// TwinCAT 3 PLC project LogToFile
// Title: Logger
// Company: FCSL
// Author: FCSL
// ProjectVersion: 0.1.0.0
// Description: Logs and tracing
// ProgramVersion: 3.1.4026.13
// libraries:
//   SPT Base Types, * (Beckhoff Automation LLC)
//   SPT Components, * (Beckhoff Automation LLC)
//   Tc2_EtherCAT, * (Beckhoff Automation GmbH)
//   Tc2_Standard, * (Beckhoff Automation GmbH)
//   Tc2_System, * (Beckhoff Automation GmbH)
//   Tc2_Utilities, * (Beckhoff Automation GmbH)
//   Tc3_BA_Common, * (Beckhoff Automation GmbH)
//   Tc3_EventLogger, * (Beckhoff Automation GmbH)
//   Tc3_JsonXml, * (Beckhoff Automation GmbH)
//   TcUnit, * (www.tcunit.org)
//   VisuSymbols,3.5.10.0,System
// project tree:
//   DUTs/ E_Result.TcDUT
//   / GlobalTextList.TcGTLO, Logger.TcTTO, PlcTask.TcTTO, Visualization Manager.TcVMO (not stored)
//   Library/Emitter/KeyValueLog/AlarmLog/ FB_AlarmLog.TcPOU
//   Library/Emitter/KeyValueLog/AuditLog/ FB_AuditLog.TcPOU (not stored)
//   Library/Emitter/KeyValueLog/ FB_FCSLBaseKeyValueLog.TcPOU (not stored)
//   Library/Listener/KeyValueLog/AlarmLog/ FB_AlarmLogListener.TcPOU
//   Library/Listener/KeyValueLog/AuditLog/ FB_AuditLogListener.TcPOU
//   Library/Listener/KeyValueLog/ FB_FCSLBaseKeyValueLogListener.TcPOU, I_KeyValueLogListener.TcIO, ST_KeyValueLogMessage.TcDUT
//   Library/Listener/ PRG_Log_Main.TcPOU
//   Library/Listener/SysLog/ FB_SysLogListener.TcPOU, I_SysLogListener.TcIO, ST_SysLogMessages.TcDUT
//   Library/Emitter/ GVL_FCSLTracing.TcGVL
//   Library/Emitter/SysLog/ E_SysLogLevel.TcDUT, FB_SysLog.TcPOU
//   LogToFile/ E_LogToFile_State.TcDUT, FB_LogToFile.TcPOU, E_LogTransmittal.TcDUT, I_Logger.TcIO (not stored), ST_LoggerSettings.TcDUT
//   TestComponents/ FB_FCSLComponentBase.TcPOU
//   TestComponents/Test Components/ FB_Test_Component.TcPOU, I_TestComponent.TcIO, PRG_TestComponents.TcPOU
//   POUs/ FB_AppendToFileDaily.TcPOU, PRG_Main.TcPOU
//   Version/ Global_Version.TcGVL
// real-time tasks:
//   TASK PlcTask: cycle T#50000us, priority 8, ADS port 350
//   TASK Logger: cycle T#10ms, priority 6, ADS port 351

CONFIGURATION LogToFile
    RESOURCE PLC ON TwinCAT3
        TASK Logger(INTERVAL := T#10ms, PRIORITY := 6);
        TASK PlcTask(INTERVAL := T#50000us, PRIORITY := 8);
        PROGRAM PRG_Log_Main WITH Logger : PRG_Log_Main;
        PROGRAM PRG_TestComponents WITH PlcTask : PRG_TestComponents;
    END_RESOURCE
END_CONFIGURATION

// ---- DUTs/E_Result.TcDUT
{attribute 'qualified_only'}
{attribute 'strict'}
{attribute 'to_string'}
TYPE E_Result :
(
	invalid := 0,
	inProgress,
	done,
	aborted
);
END_TYPE

// ---- Library/Listener/KeyValueLog/ST_KeyValueLogMessage.TcDUT
TYPE ST_KeyValueLogMessage :
    STRUCT
        timestamp 	: T_MaxString;
        k   		: T_MaxString;
        v   		: T_MaxString;	
    END_STRUCT
END_TYPE

// ---- Library/Listener/SysLog/ST_SysLogMessages.TcDUT
TYPE ST_SysLogMessages :
    STRUCT
        Timestamp : T_MaxString;
        Message   : T_MaxString;
	    LogLevel  : E_SysLogLevel;
		Source    : T_MaxString;
        Context   : T_MaxString;
        ScanCount : UDINT;
        Flags     : UDINT;
		Json   : T_MaxString;
    END_STRUCT
END_TYPE

// ---- Library/Emitter/SysLog/E_SysLogLevel.TcDUT
{attribute 'qualified_only'}
{attribute 'to_string'}
TYPE E_SysLogLevel :
(
	invalid := 0,
	testing,
	commissioning,
	production
) UDINT;
END_TYPE

// ---- LogToFile/E_LogToFile_State.TcDUT
{attribute 'qualified_only'}
{attribute 'strict'}
TYPE E_LogToFile_State :
(
	IDLE, 
	PREPARE_DATA, 
	OPEN_FILE, 
	WRITE_TO_FILE, 
	CLOSE_FILE, 
	RESET
);
END_TYPE

// ---- LogToFile/E_LogTransmittal.TcDUT
{attribute 'qualified_only'}
{attribute 'strict'}
{attribute 'to_string'}
TYPE E_LogTransmittal :
(
	invalid := 0,
	toFile,
	viaMQTT,
	viaHTTP,
	viaWS
);
END_TYPE

// ---- LogToFile/ST_LoggerSettings.TcDUT
TYPE ST_LoggerSettings :
STRUCT
	netID : STRING(20);
	filePath : T_MaxString;
	filePrefix : STRING(10);
	FileType : STRING(10);
END_STRUCT
END_TYPE

// ---- Library/Emitter/GVL_FCSLTracing.TcGVL
{attribute 'qualified_only'}
VAR_GLOBAL
	// System Log [Saved to Disk]
	sysLogLevel 		: E_SysLogLevel := E_SysLogLevel.testing;  // Current level to log to file	
	sysLog 				: FB_SysLog;
	
	// Audit Log
	auditLog 			: FB_AuditLog;
	
	//Alarm Log
	alarmLog			: FB_AlarmLog;
END_VAR

// ---- Version/Global_Version.TcGVL
{attribute 'TcGenerated'}
{attribute 'no-analysis'}
{attribute 'linkalways'}
// This function has been automatically generated from the project information.
VAR_GLOBAL CONSTANT
	{attribute 'const_non_replaced'}
	stLibVersion_Logger : ST_LibVersion := (iMajor := 0, iMinor := 1, iBuild := 0, iRevision := 0, nFlags := 0, sVersion := '0.1.0.0');
END_VAR

// ---- Library/Listener/KeyValueLog/I_KeyValueLogListener.TcIO
INTERFACE I_KeyValueLogListener

METHOD OnTraceReceived
VAR_INPUT
    message : ST_KeyValueLogMessage;
END_VAR
END_METHOD

END_INTERFACE

// ---- Library/Listener/SysLog/I_SysLogListener.TcIO
INTERFACE I_SysLogListener

METHOD OnTraceReceived
VAR_INPUT
    message : ST_SysLogMessages;
END_VAR
END_METHOD

END_INTERFACE

// ---- TestComponents/Test Components/I_TestComponent.TcIO
INTERFACE I_TestComponent EXTENDS I_BaseFB

END_INTERFACE

// ---- Library/Listener/PRG_Log_Main.TcPOU
PROGRAM PRG_Log_Main

VAR
	sysLogger 		: FB_SysLogListener;
	auditLogger		: FB_AuditLogListener;
	alarmLogger		: FB_AlarmLogListener;
END_VAR

sysLogger.CyclicLogic();
auditLogger.CyclicLogic();
alarmLogger.CyclicLogic();

END_PROGRAM

// ---- Library/Listener/SysLog/FB_SysLogListener.TcPOU
FUNCTION_BLOCK FB_SysLogListener EXTENDS FB_ListenerBase2 IMPLEMENTS I_SysLogListener
VAR
    json          			: FB_JsonDomParser; 		//Parse JSON attribute of messages
    jsonAttribute 			: STRING(10000);    		//Holds JSON attribute
    hr           			: HRESULT;         		//Signals JSON attribute was successfully read
    ipListener    			: I_SysLogListener; 	//Receives callback once message is processed
	
	fbRequestEventText 		: FB_RequestEventText;
	{attribute 'TcEncoding':='UTF-8'}
	sLastMessageText 		: STRING;
	
	
	_InitComplete			: BOOL;
	
	logger 					: FB_LogToFile;
END_VAR

METHOD CyclicLogic
IF ( NOT _initComplete ) THEN
    _initComplete := Initialize();
    RETURN;
END_IF

Execute();

logger.CyclicLogic();
END_METHOD

METHOD Initialize : BOOL
VAR
    listenerFilter 		: FB_TcEventFilter;
    hr             		: HRESULT;
END_VAR
Listener := THIS^;                                   //For callbacks on message received
ListenerFilter.Clear().EventClass.EqualTo(TC_EVENT_CLASSES.SysLog); //Filter events by tracing class
hr := Subscribe2(ListenerFilter);                    //Subscribe to retrieve defined events
IF ( SUCCEEDED(hr) ) THEN
    Initialize := TRUE;
END_IF
END_METHOD

PROPERTY Listener : I_SysLogListener
SET
ipListener := Listener;
END_SET
END_PROPERTY

METHOD OnMessageSent : Tc3_EventLogger.HRESULT
VAR_INPUT
    fbEvent 			: REFERENCE TO FB_TcEvent;
END_VAR

VAR
    message      		: ST_SysLogMessages;
    jsonDocument 		: SJsonValue;
    jsonProperty 		: SJsonValue;
	
	hasMember 			: BOOL;
END_VAR
hr := fbEvent.GetJsonAttribute(JsonAttribute, SIZEOF(JsonAttribute));

IF ( SUCCEEDED(hr) ) THEN
    jsonDocument := json.ParseDocument(JsonAttribute);

    IF ( json.HasMember(jsonDocument, 'Timestamp') ) THEN
        jsonProperty      := json.FindMember(JsonDocument, 'Timestamp');
        message.timestamp := json.GetString(JsonProperty);
    END_IF

    IF ( json.HasMember(jsonDocument, 'Message') ) THEN
        jsonProperty    := json.FindMember(jsonDocument, 'Message');
        message.message := json.GetString(jsonProperty);
    END_IF
	
	IF ( json.HasMember(jsonDocument, 'LogLevel') ) THEN
        jsonProperty      := json.FindMember(jsonDocument, 'LogLevel');
        message.logLevel := json.GetUint(jsonProperty);
    END_IF
	
    IF ( json.HasMember(jsonDocument, 'Source') ) THEN
        jsonProperty   := json.FindMember(jsonDocument, 'Source');
        message.Source := json.GetString(jsonProperty);
    END_IF

    IF ( json.HasMember(jsonDocument, 'Context') ) THEN
        jsonProperty    := json.FindMember(jsonDocument, 'Context');
        message.Context := json.GetString(jsonProperty);
    END_IF

    IF ( json.HasMember(jsonDocument, 'ScanCount') ) THEN
        jsonProperty      := json.FindMember(jsonDocument, 'ScanCount');
        message.ScanCount := json.GetUint(jsonProperty);
    END_IF

    IF ( json.HasMember(jsonDocument, 'Flags') ) THEN
        jsonProperty  := json.FindMember(jsonDocument, 'Flags');
        message.Flags := json.GetUint(jsonProperty);
    END_IF
	
    IF ( json.HasMember(jsonDocument, 'ExtendedInfo') ) THEN
        jsonProperty := json.FindMember(jsonDocument, 'ExtendedInfo');
        message.Json := json.GetString(jsonProperty);
    END_IF


    IF ( ipListener <> 0 ) THEN
        //Notify listener of message data
        ipListener.OnTraceReceived(Message);
    END_IF
END_IF

OnMessageSent := S_OK; // in order to receive more callbacks (Set <> S_OK in order to cancel the callbacks for this program cycle.)]]>
END_METHOD

METHOD OnTraceReceived
VAR_INPUT
    message 			: ST_SysLogMessages;
END_VAR

VAR
	timestamp 			: T_MaxString;
	msg   				: T_MaxString;
	logLevel  			: E_SysLogLevel;
	source    			: T_MaxString;
	context   			: T_MaxString;
	scanCount 			: UDINT;
	flags     			: UDINT;
END_VAR
// Extract relevant fields
timestamp := message.Timestamp;
msg   	  := message.Message;
logLevel  := message.LogLevel;
source    := message.Source;
context   := message.Context;
scanCount := message.ScanCount;
flags     := message.Flags;


logger.M_AddSysLog(1,msg);
END_METHOD

END_FUNCTION_BLOCK

// ---- LogToFile/FB_LogToFile.TcPOU
FUNCTION_BLOCK FB_LogToFile EXTENDS FB_CyclicFB

VAR CONSTANT
	LOG_SETTINGS 				: ST_LoggerSettings := (netID := '', filePath := 'C:\Logs\', filePrefix := 'SystemApp_', FileType := '.txt');	
	LOG_TIMEOUT 				: TIME := T#5S;
	EXPORT_INTERVAL				: TIME := T#10S;
	NEW_LINE 					: STRING(2) := '$r$n'; // Newline character
END_VAR

VAR
    ringBuffer 					: FB_StringRingBuffer;
    bufferMemory 				: ARRAY[0..5000] OF BYTE; // Adjust size as needed
	
	firstCycle 					: BOOL := TRUE;
	exportTimer					: TON;
	
	// From FB_init
    _netId 	 					: T_AmsNetId;     // Net ID for file operations
    _dirPath 					: T_MaxString;    // Directory path for the log file
	_logPrefix  				: STRING(10);     // Prefix for log file
	_fileExtension 				: STRING(10);  // File extension i.e. '.txt'
	_timeOut 					: TIME := DEFAULT_ADS_TIMEOUT;

// Params
	_execute 					: BOOL := FALSE; // Trigger for the log operation
    _data 	 					: T_MaxString; // Log entry to write

// Internal
	state 						: E_LogToFile_State;

    fileOpen  					: FB_FileOpen;
    fileClose 					: FB_FileClose;
    fileWrite 					: FB_FileWrite;

	fileRef 					: UINT := 0;       	// File handle
    risingEdge 					: R_TRIG;     // Rising edge detector for execute signal
END_VAR

VAR_OUTPUT
	smDone, smBusy, smError : BOOL;
    errId : UDINT;	 // Error ID in case of failure
END_VAR

METHOD CyclicLogic
VAR
	bufferFillPercentage: UDINT;
END_VAR
IF ( firstCycle ) THEN
	ringBuffer( pBuffer := ADR(bufferMemory), cbBuffer := SIZEOF(bufferMemory), bOverwrite := TRUE );
	firstCycle := FALSE;
	state := E_LogToFile_State.IDLE;
	RETURN;
END_IF

ringBuffer();

exportTimer(IN := TRUE, PT := EXPORT_INTERVAL);
bufferFillPercentage := (ringBuffer.cbSize * 100) / SIZEOF(bufferMemory);

IF ( ( exportTimer.Q  ) AND ( ringBuffer.nCount > 0 ) ) OR (bufferFillPercentage > 50) THEN
	//M_WriteToFile(); // Export logs when conditions are met
	_execute := TRUE;
	exportTimer(IN := FALSE); // Reset timer
ELSE
	_execute := FALSE;
END_IF;

M_StateMachine();
END_METHOD

//FB_Init is always available implicitly and it is used primarily for initialization.
//The return value is not evaluated. For a specific influence, you can also declare the
//methods explicitly and provide additional code there with the standard initialization
//code. You can evaluate the return value.
METHOD FB_Init: BOOL
VAR_INPUT
    bInitRetains: BOOL; // TRUE: the retain variables are initialized (reset warm / reset cold)
    bInCopyCode: BOOL;  // TRUE: the instance will be copied to the copy code afterward (online change)
END_VAR
_netID := LOG_SETTINGS.netID;
_dirPath := LOG_SETTINGS.filePath;
_logPrefix := LOG_SETTINGS.filePrefix;
_fileExtension := LOG_SETTINGS.FileType;
_timeOut := LOG_TIMEOUT;
END_METHOD

METHOD M_AddKeyValueLog : BOOL

VAR_INPUT
    message : ST_KeyValueLogMessage;
END_VAR

VAR
    logEntry : STRING;
END_VAR
// Concatenate severity and message
logEntry := CONCAT(message.k, ' - ');
logEntry := CONCAT(logEntry, message.v);
logEntry := CONCAT(logEntry, ' at ');
logEntry := CONCAT(logEntry, message.timestamp);

// Add log entry to ring buffer
ringBuffer.A_AddTail(putValue := logEntry);
IF ( NOT ringbuffer.bOk ) THEN
	// Handle write error (optional)END_IF;
END_IF
END_METHOD

METHOD PUBLIC M_AddSysLog : BOOL

VAR_INPUT
    severity : INT;
    message : STRING;
END_VAR

VAR
    logEntry : STRING;
END_VAR
// Concatenate severity and message
logEntry := CONCAT('Severity ', INT_TO_STRING(severity));
logEntry := CONCAT(logEntry, ': ');
logEntry := CONCAT(logEntry, message);

// Add log entry to ring buffer
ringBuffer.A_AddTail(putValue := logEntry);
IF ( NOT ringbuffer.bOk ) THEN
	// Handle write error (optional)END_IF;
END_IF
END_METHOD

METHOD PRIVATE M_CloseFile : BOOL

VAR_INPUT
	execute : BOOL;	
END_VAR
IF ( NOT execute ) THEN
	fileOpen(bExecute := FALSE);
	M_CloseFile := FALSE;
	RETURN;
END_IF

IF ( NOT fileOpen.bBusy ) THEN     
	fileClose(sNetId := _netId, hFile := fileRef, tTimeout := _timeOut);
END_IF

// Attempt to close the file
fileClose(bExecute := TRUE);

IF ( NOT M_HandleError(fileClose.bError , fileClose.nErrId) ) THEN
	fileRef := 0; // File handle
END_IF

M_CloseFile := fileClose.bBusy;
END_METHOD

METHOD PRIVATE M_HandleError : BOOL
VAR_INPUT
	check 					: BOOL;
	errorID 				: UDINT;
END_VAR
check := error;

IF check THEN
	errId := errorID;
END_IF

M_HandleError := check;
END_METHOD

METHOD PRIVATE M_OpenFile : BOOL

VAR_INPUT
	execute 				: BOOL;	
END_VAR

VAR
	getSystemTime 			: GETSYSTEMTIME; // System time function block
	fileTime 				: T_FILETIME;     // File time
	dateString 				: STRING;		// Date string for filename
	filePath 				: STRING; 	// Full log file path
END_VAR
IF ( NOT execute ) THEN
	fileOpen(bExecute := FALSE);
	M_OpenFile := FALSE;
	RETURN;
END_IF

IF ( _dirPath = '' ) THEN
   	M_HandleError(TRUE , 99);
	M_OpenFile := FALSE;
    RETURN;
END_IF

IF ( NOT fileOpen.bBusy ) THEN
	// Generate log file path with current date
	getSystemTime(timeLoDW => fileTime.dwLowDateTime, timeHiDW => fileTime.dwHighDateTime );
	dateString := SYSTEMTIME_TO_STRING(FILETIME_TO_SYSTEMTIME(fileTime));
	filepath := CONCAT(_dirPath, _logPrefix); 			// Create file path
	filePath := CONCAT(filepath, LEFT(dateString, 10)); // Add date to file path
	filePath := CONCAT(filepath, _fileExtension); 		// Add file extension to file path.
     
	fileOpen(sNetId := '', sPathName := filePath, nMode := FOPEN_MODEAPPEND, ePath := PATH_GENERIC, tTimeout := _timeOut);
END_IF

// Attempt to open the file
fileOpen(bExecute := TRUE);

IF ( NOT M_HandleError(fileOpen.bError , fileOpen.nErrId) ) THEN
	fileRef := fileOpen.hFile; // No error case
END_IF

M_OpenFile := fileOpen.bBusy;
END_METHOD

METHOD M_StateMachine

VAR
	status			: BOOL;
END_VAR
RisingEdge(CLK := _execute);

CASE state OF
    E_LogToFile_State.IDLE: // Idle state
        IF ( RisingEdge.Q ) THEN
			smDone := FALSE;
           	smBusy := TRUE;
            smError := FALSE;
            errId := 0;
		
			fileOpen(bExecute := FALSE);
			fileWrite(bExecute := FALSE);
			fileClose(bExecute := FALSE);

            state := E_LogToFile_State.OPEN_FILE;
        END_IF

    E_LogToFile_State.OPEN_FILE: // Open the file
        status := M_OpenFile(TRUE);
		IF error THEN
			state := E_LogToFile_State.CLOSE_FILE;
        ELSIF ( fileRef <> 0 ) AND ( NOT status ) THEN
			M_OpenFile(FALSE);
			state := E_LogToFile_State.PREPARE_DATA;
        END_IF
		
	E_LogToFile_State.PREPARE_DATA:
		ringBuffer.A_RemoveHead();
		_data := ringBuffer.getValue;
		
		IF ( _data <> '' ) THEN
			M_WriteToFile(FALSE, '');
			state := E_LogToFile_State.WRITE_TO_FILE;
		ELSE
			IF ( NOT fileWrite.bBusy ) THEN
				state := E_LogToFile_State.CLOSE_FILE;
			END_IF
		END_IF
		
    E_LogToFile_State.WRITE_TO_FILE: // Write to the file
		status := M_WriteToFile(execute := TRUE, inputString := _data);
		
		IF ( NOT status ) THEN
			state := E_LogToFile_State.PREPARE_DATA;
		END_IF
	
    
    E_LogToFile_State.CLOSE_FILE: // Close the file
       IF ( fileREF <> 0 ) THEN
			status :=  M_CloseFile(TRUE);
			IF ( error OR ( NOT fileWrite.bBusy ) ) THEN
				M_CloseFile(FALSE);
				state := E_LogToFile_State.RESET;
        	END_IF
		ELSE
			M_CloseFile(FALSE);
			state := E_LogToFile_State.RESET;
	   END_IF

    E_LogToFile_State.RESET: // Cleanup and reset
		smDone := TRUE;
		smBusy := FALSE;
        fileRef := 0;;
        state := E_LogToFile_State.IDLE; // Return to idle state
END_CASE
END_METHOD

METHOD PRIVATE M_WriteToFile : BOOL

VAR_INPUT
	execute : BOOL;
	inputString : STRING; // Log entry to write
END_VAR

VAR
	msgString : STRING;
END_VAR
IF ( NOT execute ) THEN
	fileOpen(bExecute := FALSE);
	fileWrite(bExecute := FALSE);
	M_WriteToFile := FALSE;
	RETURN;
END_IF

IF ( NOT fileWrite.bBusy ) THEN
	
	IF ( LEN(inputString) > (UINT_TO_INT(SIZEOF(msgString)) - LEN(NEW_LINE))) THEN
		M_HandleError( TRUE, 98);
		M_WriteToFile := FALSE;
		RETURN;
	END_IF

	msgString := CONCAT( inputString, NEW_LINE );

	// Write the message to the file
	fileWrite(sNetId := _netId, hFile := fileRef, pWriteBuff := ADR(msgString), cbWriteLen := INT_TO_UDINT(LEN(msgString)), tTimeout := +_timeOut);
END_IF

// Attempt to write the file
fileWrite(bExecute := TRUE);

IF ( M_HandleError(fileWrite.bError , fileWrite.nErrId) ) THEN
	M_WriteToFile := FALSE; // File handle
	RETURN;
END_IF

M_WriteToFile := fileWrite.bBusy;
END_METHOD

END_FUNCTION_BLOCK

// ---- Library/Listener/KeyValueLog/AuditLog/FB_AuditLogListener.TcPOU
FUNCTION_BLOCK FB_AuditLogListener EXTENDS FB_FCSLBaseKeyValueLogListener

METHOD Initialize : BOOL
VAR
    ListenerFilter : FB_TcEventFilter;
    hr             : HRESULT;
END_VAR
Listener := THIS^;                                   //For callbacks on message received
ListenerFilter.Clear().EventClass.EqualTo(TC_EVENT_CLASSES.AuditLog); //Filter events by tracing class
hr := Subscribe2(ListenerFilter);                    //Subscribe to retrieve defined events
IF ( SUCCEEDED(hr) ) THEN
    Initialize := TRUE;
END_IF
END_METHOD

END_FUNCTION_BLOCK

// ---- Library/Listener/KeyValueLog/FB_FCSLBaseKeyValueLogListener.TcPOU
FUNCTION_BLOCK FB_FCSLBaseKeyValueLogListener EXTENDS FB_ListenerBase2 IMPLEMENTS I_KeyValueLogListener
VAR
    json          			: FB_JsonDomParser; 		//Parse JSON attribute of messages
    jsonAttribute 			: STRING(10000);    		//Holds JSON attribute
    hr           			: HRESULT;         		//Signals JSON attribute was successfully read
    ipListener    			: I_KeyValueLogListener; 	//Receives callback once message is processed
	
	fbRequestEventText 		: FB_RequestEventText;
	{attribute 'TcEncoding':='UTF-8'}
	sLastMessageText 		: STRING;
	
	
	_initComplete			: BOOL;
	
	logger 					: FB_LogToFile;
END_VAR

METHOD CyclicLogic
IF NOT _InitComplete THEN
    _InitComplete := Initialize();
    RETURN;
END_IF

Execute();

logger.CyclicLogic();
END_METHOD

METHOD Initialize : BOOL
END_METHOD

PROPERTY Listener : I_KeyValueLogListener
SET
ipListener := Listener;
END_SET
END_PROPERTY

METHOD OnMessageSent : Tc3_EventLogger.HRESULT
VAR_INPUT
    fbEvent 			: REFERENCE TO FB_TcEvent;
END_VAR

VAR
    message      		: ST_KeyValueLogMessage;
    jsonDocument 		: SJsonValue;
    jsonProperty 		: SJsonValue;
	jsonExtendedInfo	: SJsonValue;
	
	bHasMember 			: BOOL;
END_VAR
hr := fbEvent.GetJsonAttribute(JsonAttribute, SIZEOF(JsonAttribute));

IF ( SUCCEEDED(hr) ) THEN
    jsonDocument := json.ParseDocument(jsonAttribute);

    IF ( json.HasMember(jsonDocument, 'Timestamp') ) THEN
        jsonProperty      := json.FindMember(jsonDocument, 'Timestamp');
        message.Timestamp := json.GetString(jsonProperty);
    END_IF

    IF ( json.HasMember(jsonDocument, 'k') ) THEN
        jsonProperty    := json.FindMember(jsonDocument, 'k');
        message.k := json.GetString(jsonProperty);
    END_IF
	
    IF ( json.HasMember(jsonDocument, 'v') ) THEN
        jsonProperty    := json.FindMember(jsonDocument, 'v');
 		message.v := json.GetString(jsonProperty);
    END_IF

    IF ( ipListener <> 0 ) THEN
        //Notify listener of message data
        ipListener.OnTraceReceived(Message);
    END_IF
END_IF

OnMessageSent := S_OK; // in order to receive more callbacks (Set <> S_OK in order to cancel the callbacks for this program cycle.)
END_METHOD

METHOD OnTraceReceived
VAR_INPUT
    message : ST_KeyValueLogMessage;
END_VAR

VAR
	timestamp			: Tc2_System.T_MaxString;
	key					: Tc2_System.T_MaxString;
	value				: Tc2_System.T_MaxString;
END_VAR
// Extract relevant fields
timestamp   := message.Timestamp;
key   := message.k;
value   := message.v;

logger.M_AddKeyValueLog(message);
END_METHOD

END_FUNCTION_BLOCK

// ---- Library/Listener/KeyValueLog/AlarmLog/FB_AlarmLogListener.TcPOU
FUNCTION_BLOCK FB_AlarmLogListener EXTENDS FB_FCSLBaseKeyValueLogListener

METHOD Initialize : BOOL
VAR
    ListenerFilter : FB_TcEventFilter;
    hr             : HRESULT;
END_VAR
Listener := THIS^;                                   //For callbacks on message received
ListenerFilter.Clear().EventClass.EqualTo(TC_EVENT_CLASSES.AlarmLog); //Filter events by tracing class
hr := Subscribe2(ListenerFilter);                    //Subscribe to retrieve defined events
IF ( SUCCEEDED(hr) ) THEN
    Initialize := TRUE;
END_IF
END_METHOD

END_FUNCTION_BLOCK

// ---- TestComponents/Test Components/PRG_TestComponents.TcPOU
PROGRAM PRG_TestComponents
VAR
	// Interfaces
	iComponent1, iComponet2, iComponet3 : I_TestComponent;	

	// Componentes
	Component_1 : FB_Test_Component := (Name := 'TC-01');
	Component_2 : FB_Test_Component := (Name := 'TC-02');
	Component_3 : FB_Test_Component := (Name := 'TC-03');

	// Test Triggers
	Trig1a, Trig1b, Trig2a, Trig2b, Trig3a, Trig3b : BOOL;
END_VAR

M_Map();

METHOD M_Map : BOOL
VAR_INPUT
END_VAR
// Map Interface
iComponent1 := Component_1;
iComponet2 := Component_2;
iComponet3 := Component_3;

// Map Parameters
Component_1.pTrig := Trig1a;
Component_1.pTrig2 := Trig1b;
Component_2.pTrig := Trig2a;
Component_2.pTrig2 := Trig2b;
Component_3.pTrig := Trig3a;
Component_3.pTrig2 := Trig3b;

// Cylic Calls
Component_1.M_CyclicLogic();
Component_2.M_CyclicLogic();
Component_3.M_CyclicLogic();
END_METHOD

END_PROGRAM

// ---- TestComponents/Test Components/FB_Test_Component.TcPOU
FUNCTION_BLOCK FB_Test_Component EXTENDS FB_FCSLComponentBase IMPLEMENTS I_TestComponent

VAR
	_trig : BOOL;
	Trig : R_TRIG;
	_trig2 : BOOL;
	Trig2 : R_TRIG;
END_VAR

VAR
	// Inputs
	MyInput AT %I* : BOOL;

	// Outputs
	MyOutput AT %Q* : BOOL;

	// HMI
//	MyComponent_HMI			: ST_ComponentMyComponent_HMI;
//	HMICommandDescendant_RT : R_TRIG;

	// Alarms
//	MyComponentAlarms : ARRAY[1..MY_COMPONENT_ALARMS_COUNT] OF FB_TcAlarm;

	// Internal variables
//	_MyVarProperty1 : BOOL;
//	_MyVarProperty2 : BOOL;
//	MyVarInternal1	: BOOL;
//	MyVarInternal2	: BOOL;

	//MyCommandFb		: MyCommandFB;// Command FB to execute something e.g. MC_MoveAbsolute
END_VAR

VAR CONSTANT
//	MY_COMPONENT_ALARMS_COUNT : UDINT := 2;
END_VAR

// NO CODE HERE!!!

//! @summary Basic component initialization logic
METHOD PRIVATE CyclicLogic

//! @description This method is called by <c>CyclicLogic()</c> as required
//! @description This method should be called cyclically by descendant function blocks by invoking <c>SUPER^.CyclicLogic()</c>. 
// Alternatively, the contents of this method could be reimplemented entirely in which case a call to this method would not be necessary.

VAR
END_VAR
IF NOT _InitComplete THEN
	_InitComplete := Initialize();
	RETURN;
END_IF

//{error 'Programming instruction - Write your custom component cyclic cogic here'}

Trig(CLK := _trig);
Trig2(CLK := _trig2);

IF Trig.Q THEN
	M_SysLog(msg := CONCAT(Name, ' : Has being triggered 1'), debug := E_SysLogLevel.testing);
END_IF

IF Trig.Q THEN
	M_AlarmLog(k := 'Raised', v := 'PT-05 warning raised, value: 5555');
END_IF
IF Trig2.Q THEN
	M_AuditLog(k := 'Login', v := 'User 1234 has logged in');
END_IF

(*
	MyCommandFb();
	IF MyCommandFB.Error THEN
		_Error	 := TRUE;
		_ErrorID := MyCommandFb.ErrorId;
	END_IF
	
	MyCommandFB.Execute := FALSE;
*)

// Component Error
//{error 'Programming instruction - Create component has error'}
//_Error	 := TRUE;
//_ErrorID := 9999;

// Component Busy
//{error 'Programming instruction - Create component is busy'}
IF FALSE THEN
	_Busy := TRUE;
ELSE
	_Busy := FALSE;
END_IF

// Call Super
SUPER^.CyclicLogic();

// Set Current Alarm Severity
// _CurrentAlarmSeverity := F_GetMaxSeverityRaised(Alarms := MyComponentAlarms, CurrentSeverity := _CurrentAlarmSeverity);
END_METHOD

(*! @summary Basic component initialization logic*)
METHOD PROTECTED Initialize : BOOL
// TODO : {error 'Programming instruction - Add code to initialize your Component'}
//M_SysLog(msg := CONCAT(Name, ' : Has being initalized'), debug := E_SysLogLevel.production);

// Call Super
Initialize := Super^.Initialize();
END_METHOD

METHOD M_CyclicLogic : BOOL
VAR_INPUT
END_VAR
CyclicLogic();
//test
END_METHOD

PROPERTY pTrig : BOOL
GET
pTrig := _trig;
END_GET
SET
_trig := pTrig;
END_SET
END_PROPERTY

PROPERTY pTrig2 : BOOL
GET
pTrig2 := _trig2;
END_GET
SET
_trig2 := pTrig2;
END_SET
END_PROPERTY

END_FUNCTION_BLOCK

// ---- TestComponents/FB_FCSLComponentBase.TcPOU
FUNCTION_BLOCK FB_FCSLComponentBase EXTENDS FB_ComponentBase

VAR

END_VAR

METHOD M_AlarmLog : HRESULT

VAR_INPUT
	k : T_MaxString;
	v : T_MaxString;
END_VAR
GVL_FCSLTracing.alarmLog.M_AddEntry(k := k, v := v);

M_AlarmLog := S_OK;
END_METHOD

METHOD M_AuditLog : HRESULT

VAR_INPUT
	k : T_MaxString;
	v : T_MaxString;
END_VAR
GVL_FCSLTracing.auditLog.M_AddEntry(k := k, v := v);

M_AuditLog := S_OK;
END_METHOD

METHOD M_SysLog : HRESULT

VAR_INPUT
	msg 			: T_MaxString;
	debug 			: E_SysLogLevel;
END_VAR

VAR
	debugString 	: STRING;
	debugINT 		: UDINT;
	json 			: T_MaxString;	
END_VAR
IF ( debug = E_SysLogLevel.invalid ) THEN
	RETURN;
END_IF

// Send log entry
GVL_FCSLTracing.sysLog.M_AddEntry(
    Source := InstancePath, 
    Message := msg, 
    logLevel := debug, 
    Flags := 0
);

// Return success
M_SysLog := S_OK;
END_METHOD

END_FUNCTION_BLOCK

// ---- Library/Emitter/SysLog/FB_SysLog.TcPOU
FUNCTION_BLOCK FB_SysLog
VAR
	event						 	: FB_TcMessage;
	jsonParser					 	: FB_JsonDomParser;
	exParser 				 		: FB_JsonDomParser;
	timeFormatter				 	: FB_FormatString;
	messagesSentThisScan		 	: UDINT;
	previousAddEntrySource		 	: T_MaxString;
	previousAddEntryMessage	 		: T_MaxString;
	previousAddEntryFlags		 	: UDINT;
	previousAddEntryJsonSource	 	: T_MaxString;
	previousAddEntryJsonMessage 	: T_MaxString;
	previousAddEntryJsonFlags	 	: UDINT;
	previousAddEntryJson		 	: T_MaxString;
	initComplete				 	: BOOL := FALSE;
END_VAR

//FB_Init is always available implicitly and it is used primarily for initialization.
//The return value is not evaluated. For a specific influence, you can also declare the
//methods explicitly and provide additional code there with the standard initialization
//code. You can evaluate the return value.
METHOD FB_Init: BOOL
VAR_INPUT
    bInitRetains: BOOL; // TRUE: the retain variables are initialized (reset warm / reset cold)
    bInCopyCode: BOOL;  // TRUE: the instance will be copied to the copy code afterward (online change)   
END_VAR

VAR
	hr : HRESULT;
END_VAR
//	IF SUCCEEDED(Event.CreateEx(TC_EVENTS.Tracing.TraceEvent, 0)) THEN
{analysis -15}
IF ( NOT Event.EqualsToEventEntryEx(TC_EVENTS.Tracing.TraceEvent) ) THEN
	IF ( SUCCEEDED(Event.CreateEx(TC_EVENTS.SysLog.Logger, 0)) ) THEN
		InitComplete := TRUE;
	END_IF
ELSE
	InitComplete := TRUE;
END_IF
END_METHOD

METHOD PRIVATE M_AddContext

VAR_INPUT
	json 			: SJsonValue;
	message 		: REFERENCE TO T_MaxString;
	logLevel 		: E_SysLogLevel;
	source 			: STRING;
	flags  			: UDINT;
END_VAR

VAR
	// Time 
	CurrentDCTime : DCTIMESTRUCT;
	Task : T_MaxString;
	CycleCount : UDINT;
END_VAR
//Collect Properties
currentDCTime := DCTIME64_TO_DCTIMESTRUCT(F_GetActualDcTime64());
TimeFormatter(
    sFormat := '%2.2d:%2.2d:%2.2d.%3.3d%3.3d',
    arg1    := F_WORD(currentDCTime.wHour),
    arg2    := F_WORD(currentDCTime.wMinute),
    arg3    := F_WORD(currentDCTime.wSecond),
    arg4    := F_WORD(currentDCTime.wMilliseconds),
    arg5    := F_WORD(currentDCTime.wMicroseconds),	
    bError  => ,    // If there's a formatting error, this is TRUE
    nErrId  =>      // Error ID if bError=TRUE
);		
task := TwinCAT_SystemInfoVarList._TaskInfo[GETCURTASKINDEXEX()].TaskName;
cycleCount := TwinCAT_SystemInfoVarList._TaskInfo[GETCURTASKINDEXEX()].CycleCount;

event.ipArguments.Clear().AddString(Message);

// Pass properties to Json extnsion for logging.
jsonParser.AddStringMember(json, 'Timestamp', timeFormatter.sOut);
jsonParser.AddStringMember(json, 'Message', message);
jsonParser.AddUIntMember(json, 'LogLevel', logLevel);
jsonParser.AddStringMember(json, 'Source', source);
jsonParser.AddStringMember(json, 'Context', task);
jsonParser.AddUint64Member(json, 'ScanCount', cycleCount);
jsonParser.AddUint64Member(json, 'Flags', flags);
END_METHOD

METHOD M_AddEntry : BOOL
VAR_INPUT
	source				: T_MaxString;
	message 			: T_MaxString;
	logLevel 			: E_SysLogLevel;
	flags				: UDINT;
END_VAR

VAR
	document	  		: SJsonValue;
	jsonAttribute 		: T_MaxString;
END_VAR
IF ( NOT InitComplete )THEN
	RETURN;
END_IF

{analysis -62}
IF ( NOT pTracingAllowed ) THEN
	{analysis -90}
	RETURN;
END_IF

IF ( NOT Parameters_Tracing.ALLOW_DUPLICATE_SEQUENTIAL_MESSAGES ) THEN
	IF (Source = previousAddEntrySource) AND (Message = previousAddEntryMessage) AND (Flags = previousAddEntryFlags) THEN
		//This message is identical to the last message sent--ignore
		RETURN;
	END_IF
END_IF

// Create JSON, add Context and add to Event
document := jsonParser.NewDocument();
M_AddContext(JSON := document, message := message, logLevel := logLevel, source := source, flags := flags);
jsonAttribute := jsonParser.GetJson(document);
event.SetJsonAttribute(jsonAttribute);

// Send Event
Event.Send(0);


// Tidy up
MessagesSentThisScan := MessagesSentThisScan + 1;
MEMSET(ADR(previousAddEntrySource), 0, SIZEOF(T_MaxString));
MEMSET(ADR(previousAddEntryMessage), 0, SIZEOF(T_MaxString));
previousAddEntrySource	 := Source;
previousAddEntryMessage := Message;
previousAddEntryFlags	 := Flags;
END_METHOD

PROPERTY pTracingAllowed : BOOL
GET
VAR_INST
	LastScanCount  : UDINT;
	MissedMessages : UDINT;
	Throttled	   : BOOL;
END_VAR

VAR
	ThrottledNotificationString : T_MaxString;
END_VAR
{analysis -62}
IF NOT Parameters_Tracing.TRACING_ENABLED THEN
	pTracingAllowed := FALSE;
	RETURN;
END_IF

IF TwinCAT_SystemInfoVarList._TaskInfo[GETCURTASKINDEXEX()].CycleCount = LastScanCount THEN
	//Trying to send multiple messages in same scan
	IF Throttled THEN
		MissedMessages := MissedMessages + 1;
		RETURN;
	ELSIF MessagesSentThisScan >= Parameters_Tracing.MAX_LOG_ENTRIES_PER_SCAN AND NOT Throttled THEN
		//Need to throttle messsage queue
		Event.ipArguments.Clear().AddString('Too many messages sent in single scan; tracing throttled.');
		Event.Send(0);
		MissedMessages := MissedMessages + 1;
		Throttled	   := TRUE;
		pTracingAllowed := FALSE;
		RETURN;
	ELSE
		pTracingAllowed := TRUE;
	END_IF
ELSE
	IF Throttled THEN
		ThrottledNotificationString := CONCAT('Missed ', CONCAT(TO_STRING(MissedMessages), ' throttled messages previously.'));
		Event.ipArguments.Clear().AddString(ThrottledNotificationString);
		Event.Send(0);
		MissedMessages := 0;
	END_IF

	LastScanCount		 := TwinCAT_SystemInfoVarList._TaskInfo[GETCURTASKINDEXEX()].CycleCount;
	MessagesSentThisScan := 0;
	Throttled			 := FALSE;
	pTracingAllowed		 := TRUE;
END_IF
END_GET
END_PROPERTY

END_FUNCTION_BLOCK

// ---- Library/Emitter/KeyValueLog/AlarmLog/FB_AlarmLog.TcPOU
FUNCTION_BLOCK FB_AlarmLog EXTENDS FB_FCSLBaseKeyValueLog

//FB_Init is always available implicitly and it is used primarily for initialization.
//The return value is not evaluated. For a specific influence, you can also declare the
//methods explicitly and provide additional code there with the standard initialization
//code. You can evaluate the return value.
METHOD FB_Init: BOOL
VAR_INPUT
    bInitRetains: BOOL; // TRUE: the retain variables are initialized (reset warm / reset cold)
    bInCopyCode: BOOL;  // TRUE: the instance will be copied to the copy code afterward (online change)   
END_VAR

VAR
	hr : HRESULT;
END_VAR
//	IF SUCCEEDED(Event.CreateEx(TC_EVENTS.Tracing.TraceEvent, 0)) THEN
{analysis -15}
IF ( NOT Event.EqualsToEventEntryEx(TC_EVENTS.Tracing.TraceEvent) ) THEN
	IF ( SUCCEEDED(Event.CreateEx(TC_EVENTS.AlarmLog.Logger, 0)) ) THEN
		initComplete := TRUE;
	END_IF
ELSE
	initComplete := TRUE;
END_IF
END_METHOD

END_FUNCTION_BLOCK

// ---- POUs/FB_AppendToFileDaily.TcPOU
FUNCTION_BLOCK FB_AppendToFileDaily
VAR_INPUT
    sNetId : T_AmsNetId;     // Net ID for file operations
    sPath  : T_MaxString;    // Directory path for the log file
    inputString : STRING(255); // Log entry to write
    bExecute : BOOL;         // Trigger for logging
    tTimeOut : TIME := DEFAULT_ADS_TIMEOUT;
END_VAR
VAR_OUTPUT
    bBusy : BOOL;            // TRUE if logging is in progress
    bError : BOOL;           // TRUE if an error occurs
    nErrId : UDINT;          // Error ID in case of failure
END_VAR
VAR
    fbFileOpen : FB_FileOpen;
    fbFileClose : FB_FileClose;
    fbFileWrite : FB_FileWrite;
 	fbGetSystemTime : GETSYSTEMTIME; // System time function block
 	fileTime : T_FILETIME;     // File time
  
    hFile : UINT := 0;       // File handle
    sFilePath : STRING(255); // Full log file path
    sTime : STRING;          // Date string for filename
    sNewLine : STRING(2) := '$r$n'; // Newline character
    msgString : STRING(255); // Full message with newline
    Step : DWORD := 0;       // State machine step
    RisingEdge : R_TRIG;     // Rising edge detector for execute signal
END_VAR


RisingEdge(CLK := bExecute);

CASE Step OF
    0: // Idle state
        IF RisingEdge.Q THEN
            bBusy := TRUE;
            bError := FALSE;
            nErrId := 0;
            hFile := 0;
          	
            // Generate log file path with current date
            fbGetSystemTime(timeLoDW=>fileTime.dwLowDateTime, timeHiDW=>fileTime.dwHighDateTime );
	    	sTime := SYSTEMTIME_TO_STRING(FILETIME_TO_SYSTEMTIME(fileTime));
        	sFilePath := CONCAT('C:\Logs\', CONCAT(LEFT(sTime, 10), '.txt'));
     
            Step := 1;
        END_IF

    1: // Open or create the log file
        fbFileOpen(bExecute := FALSE);
        fbFileOpen(sNetId := sNetId, sPathName := sFilePath, nMode := FOPEN_MODEAPPEND, ePath := PATH_GENERIC, tTimeout := tTimeOut, bExecute := TRUE);
        Step := 2;

    2: // Wait for file open
        fbFileOpen(bExecute := TRUE);
        IF NOT fbFileOpen.bBusy THEN
            IF fbFileOpen.bError THEN
                nErrId := fbFileOpen.nErrId;
                bError := TRUE;
                Step := 50; // Cleanup
            ELSE
                hFile := fbFileOpen.hFile;
                Step := 3;
            END_IF
        END_IF

    3: // Prepare the message to write
        msgString := CONCAT(sNewLine, inputString);
        Step := 4;

    4: // Write the message to the file
        fbFileWrite(bExecute := FALSE);
        fbFileWrite(sNetId := sNetId, hFile := hFile, pWriteBuff := ADR(msgString), cbWriteLen := LEN(msgString), bExecute := TRUE, tTimeout := tTimeOut);
        Step := 5;

    5: // Wait for write completion
        fbFileWrite(bExecute := TRUE);
        IF NOT fbFileWrite.bBusy THEN
            IF fbFileWrite.bError THEN
                nErrId := fbFileWrite.nErrId;
                bError := TRUE;
                Step := 50; // Cleanup
            ELSE
                Step := 30; // Close file after writing
            END_IF
        END_IF

    30: // Close the file
        fbFileClose(bExecute := FALSE);
        fbFileClose(sNetId := sNetId, hFile := hFile, bExecute := TRUE, tTimeout := tTimeOut);
        Step := 31;

    31: // Wait for file close
        fbFileClose(bExecute := TRUE);
        IF NOT fbFileClose.bBusy THEN
            IF fbFileClose.bError THEN
                nErrId := fbFileClose.nErrId;
                bError := TRUE;
            END_IF
            Step := 50; // Final cleanup
        END_IF

    50: // Cleanup and reset
        hFile := 0;
        bBusy := FALSE;
        Step := 0; // Return to idle state
END_CASE

END_FUNCTION_BLOCK

// ---- POUs/PRG_Main.TcPOU
PROGRAM PRG_Main
VAR
    fbLogger : FB_AppendToFileDaily;
    bLog : BOOL := TRUE; // Trigger to log data
END_VAR

IF bLog THEN
    fbLogger(sNetId := '', sPath := 'C:\Logs\', inputString := 'This is a test log entry 2222', bExecute := TRUE);
    
    IF NOT fbLogger.bBusy THEN
        IF fbLogger.bError THEN
            // Handle error
        ELSE
            // Log successfully written
        END_IF
        bLog := FALSE; // Reset trigger
		fbLogger(bExecute := FALSE);
    END_IF
END_IF

END_PROGRAM
